(* CODESYS project CtaAppEinsatzDiagramm_2.0.0.0.library
   Description: Einsatzdiagramm Library der CTA
   Version: 2.0.0.0
   Title: CtaAppEinsatzDiagramm
   Author: SIS
   DocFormat: reStructuredText
   LanguageModelAttribute: qualified-access-only
   Placeholder: CtaAppEinsatzDiagramm
   CompiledLibraryCompatibilityVersion: CODESYS V3.5 SP16 Patch 3
   Company: CTA
   DefaultNamespace: CtaAppEinsatzDiagramm

Project tree, tasks and I/O mapping:
  libraries: Standard, 3.5.18.0 (System); CtaAppBmk, 2.0.0.0 (CTA); CtaAppReport, 2.0.0.0 (CTA); CtaSysConfig, 2.0.0.0 (CTA); CtaAppHysterese, 1.0.0.0 (CTA); VisuElemBase, 4.7.0.0 (System); VisuDialogs, * (System); CtaVisSymbols, 2.0.0.0 (CTA); CtaVisUser, 1.0.0.0 (CTA); VisuSymbols, 4.5.0.0 (System); CtaVisApps, 1.0.0.0 (CTA); CtaVisHelp, 1.0.0.0 (CTA)
  40 Visualizations/
    EINSATZGRENZE/
      visualisation VIS_EINSATZGRENZE
      visualisation VIS_EINSATZGRENZE_ITF
      visualisation VIS_EINSATZGRENZE_QUERRY
      DIALOG/
        visualisation DIA_EINSATZGRENZE
        visualisation VIS_DIA_EINSATZGRENZE
        visualisation VIS_DIA_EINSATZGRENZE_ITF
  30 Program Organization Units/
    Einsatzgrenzen/
      function block fbEinsatzgrenze [ST]: actDiagrammPaint, actAktualPoint, actBerrechnung, actÜberwachung, actReport, actConfigFile, proTHIS_REF
  00000000-0000-0000-0000-000000000000|D:\CoDeSys\LibrariesV3\trunk\Intern\CAA\CAA Template\3.4.0.0 draft\Placeholder.xml
  00000000-0000-0000-0000-000000000000|D:\CoDeSys\LibrariesV3\trunk\Intern\CAA\CAA Template\3.2.0.3 draft\Prefix.pdf
  00000000-0000-0000-0000-000000000000|D:\CoDeSys\LibrariesV3\trunk\Intern\CAA\CAA Template\3.5.2.0 draft\Placeholder.xml
  20 Structs/
    Einsatzgrenze/
      data type scParameterEinsatzgrenze
      Paint/
        data type scLinePoint
        data type scDiagrammSizePaint
      Parameter/
        data type scSlopValue1
        data type scSlopValue2
        data type scSlopValue3
        data type scSlopValue4
        data type scSlopValue5
        data type scSlopValue6
        data type scDiagrammSize
        data type scErrorWarning
  50 Images/
  10 Documenation/
    global variables VersionHistory
    global variables readMe
  21 Interface/
    interface ITF_EINSATZGRENZE: proTHIS_REF
  11 Library Parameter/
    global variables Parameter
  12 Konstanten/
    global variables GlobalKonstant
  60 Textlisten/
    text list Error
    text list Info
    text list Warnung
  13 Globale Variablen/
  text list GlobalTextList
  5ce3da45-db07-42e7-a21c-a00fff4ed8f6|C:\Users\sis\Downloads\dip-switch.svg
  5ce3da45-db07-42e7-a21c-a00fff4ed8f6|C:\Users\sis\Downloads\lightning-bolt-circle.svg
  5ce3da45-db07-42e7-a21c-a00fff4ed8f6|C:\Users\sis\Downloads\sine-wave.svg
  5ce3da45-db07-42e7-a21c-a00fff4ed8f6|C:\Users\sis\Downloads\eye.svg
  5ce3da45-db07-42e7-a21c-a00fff4ed8f6|C:\Users\sis\Downloads\lan.svg
*)

// 20 Structs/Einsatzgrenze/scParameterEinsatzgrenze
TYPE scParameterEinsatzgrenze :
    STRUCT
        scDiagrammSize              :   scDiagrammSize;
        fbrMinTc					:	CtaSysConfig.fbREAL;							        // Minimale Kondensationstemperatur [°C] 
        fbrMaxTc					:	CtaSysConfig.fbREAL;							        // Maximale Kondensationstemperatur [°C] 
        fbrMinTo					:	CtaSysConfig.fbREAL;							        // Minimale Verdampfungstemperatur  [°C]
        fbrMaxTo					:	CtaSysConfig.fbREAL; 							        // Maximale Verdampfungstemperatur  [°C]             
        scSlopValue1                :   scSlopValue1;         
        scSlopValue2                :   scSlopValue2;
        scSlopValue3                :   scSlopValue3;
        scSlopValue4                :   scSlopValue4;
        scSlopValue5                :   scSlopValue5;
        scSlopValue6                :   scSlopValue6;        
        scErrorWarning              :   scErrorWarning; 
    END_STRUCT
END_TYPE

// 20 Structs/Einsatzgrenze/Paint/scLinePoint
TYPE scLinePoint :
    STRUCT
        rP1X        :   REAL;
        rP1Y        :   REAL;      
    END_STRUCT
END_TYPE

// 20 Structs/Einsatzgrenze/Paint/scDiagrammSizePaint
TYPE scDiagrammSizePaint :
    STRUCT
        rYMax   :   REAL;
        rYMin   :   REAL;
        rXMax   :   REAL;
        rXMin   :   REAL;    
    END_STRUCT
END_TYPE

// 20 Structs/Einsatzgrenze/Parameter/scSlopValue1
TYPE scSlopValue1 :
    STRUCT
        fbrTcL			    :	CtaSysConfig.fbREAL;							        // Punkt  1 Kompressor-Auslegungsdiagramm [°C] 
        fbrT0L              :   CtaSysConfig.fbREAL;	                                // Punkt  2 Kompressor-Auslegungsdiagramm [°C]
        fbrT0R  		    :	CtaSysConfig.fbREAL;							        // Punkt  3 Kompressor-Auslegungsdiagramm [°C]        
    END_STRUCT
END_TYPE

// 20 Structs/Einsatzgrenze/Parameter/scSlopValue2
TYPE scSlopValue2 :
    STRUCT
        fbrTcR			    :	CtaSysConfig.fbREAL;							        // Punkt  4 Kompressor-Auslegungsdiagramm [°C] 
        fbrT0R  		    :	CtaSysConfig.fbREAL;							        // Punkt  5 Kompressor-Auslegungsdiagramm [°C]        
    END_STRUCT
END_TYPE

// 20 Structs/Einsatzgrenze/Parameter/scSlopValue3
TYPE scSlopValue3 :
    STRUCT
        fbrTcU			    :	CtaSysConfig.fbREAL;							        // Punkt  6 Kompressor-Auslegungsdiagramm [°C] 
    END_STRUCT
END_TYPE

// 20 Structs/Einsatzgrenze/Parameter/scSlopValue4
TYPE scSlopValue4 :
    STRUCT
        fbrTcL			    :	CtaSysConfig.fbREAL;							        // Punkt  7 Kompressor-Auslegungsdiagramm [°C]         
    END_STRUCT
END_TYPE

// 20 Structs/Einsatzgrenze/Parameter/scSlopValue5
TYPE scSlopValue5 :
    STRUCT
        fbrT0L			    :	CtaSysConfig.fbREAL;							        // Punkt  8 Kompressor-Auslegungsdiagramm [°C] 
        fbrT0R  			:	CtaSysConfig.fbREAL;							        // Punkt  9 Kompressor-Auslegungsdiagramm [°C]                
    END_STRUCT
END_TYPE

// 20 Structs/Einsatzgrenze/Parameter/scSlopValue6
TYPE scSlopValue6 :
    STRUCT
        fbrTcO			    :	CtaSysConfig.fbREAL;							        // Punkt 10 Kompressor-Auslegungsdiagramm [°C]                 
    END_STRUCT
END_TYPE

// 20 Structs/Einsatzgrenze/Parameter/scDiagrammSize
TYPE scDiagrammSize :
    STRUCT
        fbrYMax   :   CtaSysConfig.fbREAL;
        fbrYMin   :   CtaSysConfig.fbREAL;
        fbrXMax   :   CtaSysConfig.fbREAL;
        fbrXMin   :   CtaSysConfig.fbREAL;    
    END_STRUCT
END_TYPE

// 20 Structs/Einsatzgrenze/Parameter/scErrorWarning
TYPE scErrorWarning :
    STRUCT
        fbxEnEW1          :   CtaSysConfig.fbBOOL;
        fbxEnEW2          :   CtaSysConfig.fbBOOL;
        fbxEnEW3          :   CtaSysConfig.fbBOOL;
        fbxEnEW4          :   CtaSysConfig.fbBOOL;
        fbxEnEW5          :   CtaSysConfig.fbBOOL;
        fbxEnEW6          :   CtaSysConfig.fbBOOL;
        fbxEnEW7          :   CtaSysConfig.fbBOOL;
        fbtDelayWarning   :   CtaSysConfig.fbTIME;
        fbiAnzError       :   CtaSysConfig.fbINT;
        fbtDelayError     :   CtaSysConfig.fbTIME;
        fbtCountReset     :   CtaSysConfig.fbTIME;
    END_STRUCT
END_TYPE

// 10 Documenation/VersionHistory
(* 

.. image:: ../../Images/CTA_Logo.jpg
   :align: right
   :width: 15% 

**Vorlage**   


============ =========== =========== ============================================
**Date**     **Version** **Author**  **Change**
------------ ----------- ----------- --------------------------------------------
04.03.2021   0.0.0.0     SIS         Vorlage erstellt

============ =========== =========== ============================================


*)
VAR_GLOBAL
    stInfo : STRING:= '0.0.0.0, Vorlage, CTA';
END_VAR

// 10 Documenation/readMe
(*

**ReadMe**
 
|	**Empfehlung**
|
|	Bibliothek CtaAppVerdichter zur Ansteuerung von Verdichtern
|	Instanzieren Sie den CtaAppVerdichter.fbVerdichter in ihrem Funktionsbaustein oder POU beispielsweise als fbVerdiX. (X = Nr.)
|	Instanzieren Sie den CtaAppVerdichter.fbEinsatzgrenze in ihrem Funktionsbaustein oder POU beispielsweise als fbVerdiXEinsatzGr. (X = Nr des Verdicheters)
|	Deklarieren Sie die Struktur Variable welche als Parameter und zur ansteuerung dienen wie im Code beispiel.
|  
| *Beispiel* 

+-----------------------+---------------------------------------------------------------------------------------------------------------------------------------------------------------------------------------------------------------------------------------------------------------------------------------------------------------------------------------------------------------------------------------------------------------------------------------+
| Beschreibung          |  Code                                                                                                                                                                                                                                                                                                                                                                                                                                 |
+=======================+=======================================================================================================================================================================================================================================================================================================================================================================================================================================+
| Pou oder SmFb         | .. code-block:: codesys                                                                                                                                                                                                                                                                                                                                                                                                               |
|                       |                                                                                                                                                                                                                                                                                                                                                                                                                                       |
|                       |	// Deklaration als VAR im POU oder dem selbsterstellten Funktionsbaustein                                                                                                                                                                                                                                                                                                                                                       	|
|                       |   VAR   																																																																																																								|
|						|	    (*Einsatzgrenze Verdichter1*)																																																		 																																															|
|						|		fbVerdi1EinsatzGr	: CtaAppVerdichter.fbEinsatzgrenze;                                                                                                                                                                                                                                                                                                                                                              			|
| 						|	END_VAR                                                                                                                                                                                                                                                                                                                                                                                                                         	|
+-----------------------+---------------------------------------------------------------------------------------------------------------------------------------------------------------------------------------------------------------------------------------------------------------------------------------------------------------------------------------------------------------------------------------------------------------------------------------+
| Code für Init         | .. code-block:: codesys                                                                                                                                                                                                                                                                                                                                                                                                               |
|                       |   																																																																																																									|
| 						|	// Kopieren des nachfolgenden Codes in eine Action zur Initialisierung der Parameter. Zum Beispiel actConfig.																																																																														|
|                       |	{region "Parameter Einsatzgrenzen Verdichter1"}                                                                                                                                                                                                                                                                                                                                                                                     |
| 						|		(*Diagrammgrösse*)																																																																																																				|
|						|		fbVerdi1EinsatzGr.scParaData.scDiagrammSize.fbrYMax               		(_wertInit :=   0.0									, _minInit :=		, _maxInit :=		);		//P1 Diagrammgrösse Y Achse Max																																																						|
|						|		fbVerdi1EinsatzGr.scParaData.scDiagrammSize.fbrYMin						(_wertInit :=   0.0									, _minInit :=		, _maxInit :=		);		//P2 Diagrammgrösse Y Achse Min																																																						|
|						|		fbVerdi1EinsatzGr.scParaData.scDiagrammSize.fbrXMax						(_wertInit :=   0.0									, _minInit :=		, _maxInit :=		);		//P3 Diagrammgrösse X Achse Max																																																						|
|						|		fbVerdi1EinsatzGr.scParaData.scDiagrammSize.fbrXMin						(_wertInit :=   0.0									, _minInit :=		, _maxInit :=		);		//P4 Diagrammgrösse X Achse Min																																																						|
|						|		(*Min Max Tc & To*)																																																		 																																																		|
|						|		fbVerdi1EinsatzGr.scParaData.fbrMinTc									(_wertInit :=   0.0									, _minInit :=		, _maxInit :=		);		//P5 Max Tc																																																											|
|						|		fbVerdi1EinsatzGr.scParaData.fbrMaxTc									(_wertInit :=   0.0									, _minInit :=		, _maxInit :=		);		//P6 Min Tc																																																											|
|						|		fbVerdi1EinsatzGr.scParaData.fbrMinTo									(_wertInit :=   0.0									, _minInit :=		, _maxInit :=		);		//P7 Max To																																																											|
|						|		fbVerdi1EinsatzGr.scParaData.fbrMaxTo									(_wertInit :=   0.0									, _minInit :=		, _maxInit :=		);		//P8 Min To																																																											|
|						|		(*Slop Value 1*)																																																		 																																																		|
|						|		fbVerdi1EinsatzGr.scParaData.scSlopValue1.fbrTcL						(_wertInit :=   0.0									, _minInit :=		, _maxInit :=		);		//P9 Slop Value 1 Tc Links																	    																																					|
|						|		fbVerdi1EinsatzGr.scParaData.scSlopValue1.fbrT0L						(_wertInit :=   0.0									, _minInit :=		, _maxInit :=		);		//P10 Slop Value 1 To Links																												    																										|
|						|		fbVerdi1EinsatzGr.scParaData.scSlopValue1.fbrT0R						(_wertInit :=   0.0									, _minInit :=		, _maxInit :=		);		//P11 Slop Value 1 To Rechts																											    																										|
|						|		(*Slop Value 2*)																																																										 																																	  									|
|						|		fbVerdi1EinsatzGr.scParaData.scSlopValue2.fbrTcR						(_wertInit :=   0.0									, _minInit :=		, _maxInit :=		);		//P12 Slop Value 2 Tc Rechts																    																																					|
|						|		fbVerdi1EinsatzGr.scParaData.scSlopValue2.fbrT0R						(_wertInit :=   0.0									, _minInit :=		, _maxInit :=		);		//P13 Slop Value 2 To Rechts																																								   	 													|
|						|		(*Slop Value 3*)																																																											 																																							    	|
|						|		fbVerdi1EinsatzGr.scParaData.scSlopValue3.fbrTcU						(_wertInit :=   0.0									, _minInit :=		, _maxInit :=		);		//P14 Slop Value 3 Tc Unten																														    																								|
|						|		(*Slop Value 4*)																																																											 																																							    	|
|						|		fbVerdi1EinsatzGr.scParaData.scSlopValue4.fbrTcL						(_wertInit :=   0.0									, _minInit :=		, _maxInit :=		);		//P15 Slop Value 4 Tc Links																																				    																		|
|						|		(*Slop Value 5*)																																																		 																																																		|
|						|		fbVerdi1EinsatzGr.scParaData.scSlopValue5.fbrT0L						(_wertInit :=   0.0									, _minInit :=		, _maxInit :=		);		//P16 Slop Value 5 To Links																																		    																				|
|						|		fbVerdi1EinsatzGr.scParaData.scSlopValue5.fbrT0R						(_wertInit :=   0.0									, _minInit :=		, _maxInit :=		);		//P17 Slop Value 5 To Rechts																																		    																			|
|						|		(*Slop Value 6*)																																																		 																																																		|
|						|		fbVerdi1EinsatzGr.scParaData.scSlopValue6.fbrTcO						(_wertInit :=   0.0									, _minInit :=		, _maxInit :=		);		//P18 Slop Value 6 Tc Oben																																																							|
|						|		(*Error & Warnungen*)																																																																																																		    |
|						|		fbVerdi1EinsatzGr.scParaData.scErrorWarning.fbxEnEW1					(_wertInit := FALSE																			);		//P19 Überwachung Slop Value 1																																	    																				|
|						|		fbVerdi1EinsatzGr.scParaData.scErrorWarning.fbxEnEW2					(_wertInit := FALSE																			);		//P20 Überwachung Slop Value 2																																										    											|
|						|		fbVerdi1EinsatzGr.scParaData.scErrorWarning.fbxEnEW3					(_wertInit := FALSE																			);		//P21 Überwachung Slop Value 3																														   																								|
|						|		fbVerdi1EinsatzGr.scParaData.scErrorWarning.fbxEnEW4					(_wertInit := FALSE																			);		//P22 Überwachung Slop Value 4																																								    													|
|						|		fbVerdi1EinsatzGr.scParaData.scErrorWarning.fbxEnEW5					(_wertInit := FALSE																			);		//P23 Überwachung Slop Value 5				   																																																		|
|						|		fbVerdi1EinsatzGr.scParaData.scErrorWarning.fbxEnEW6					(_wertInit := FALSE																			);		//P24 Überwachung Slop Value 6																						   																																|
|						|		fbVerdi1EinsatzGr.scParaData.scErrorWarning.fbxEnEW7					(_wertInit := FALSE																			);		//P25 Überwachung Slop Value 7														    																																							|
|						|		fbVerdi1EinsatzGr.scParaData.scErrorWarning.fbtDelayWarning				(_wertInit := T#00S									, _minInit :=		, _maxInit :=		);		//P26 Warnungsverzögerung																																																							|
|						|		fbVerdi1EinsatzGr.scParaData.scErrorWarning.fbiAnzError					(_wertInit :=     0									, _minInit :=		, _maxInit :=		);		//P27 Anzahl Error Autoquittierungen																																																				|
|						|		fbVerdi1EinsatzGr.scParaData.scErrorWarning.fbtDelayError				(_wertInit := T#00S									, _minInit :=	    , _maxInit :=		);		//P28 Errorverzögerung																																																								|
|						|		fbVerdi1EinsatzGr.scParaData.scErrorWarning.fbtCountReset				(_wertInit := T#00S									, _minInit :=		, _maxInit :=		);		//P29 Reset des Zähler nach t																																																						|
|						|	{endregion}                                             	                                                                                                         																																																																|
+-----------------------+---------------------------------------------------------------------------------------------------------------------------------------------------------------------------------------------------------------------------------------------------------------------------------------------------------------------------------------------------------------------------------------------------------------------------------------+
*)                                                                                                                                                                                                                                                                                                                                                                                                                                                               
 VAR_GLOBAL                                                                                                                                                                                                                                                                                                                                                                                                                                                      
    xReadMeDone              :   BOOL;                                                                                                                                                                                                                                                                                                                                                                                                                           
END_VAR

// 11 Library Parameter/Parameter
{attribute 'qualified_only'}
VAR_GLOBAL CONSTANT
    iMaxVerdichter :   INT   := 60;         // Maximale Anzahl verwendeter AT-Bausteine    
END_VAR

// 12 Konstanten/GlobalKonstant
{attribute 'qualified_only'}
VAR_GLOBAL CONSTANT 	
	stReportTextListError   : CtaAppReport.stReportTextList := 'CtaAppEinsatzDiagramm.Error';
	stReportTextListWarning : CtaAppReport.stReportTextList := 'CtaAppEinsatzDiagramm.Warnung';
	stReportTextListInfo    : CtaAppReport.stReportTextList := 'CtaAppEinsatzDiagramm.Info';	
END_VAR

// 30 Program Organization Units/Einsatzgrenzen/fbEinsatzgrenze
FUNCTION_BLOCK fbEinsatzgrenze IMPLEMENTS ITF_EINSATZGRENZE
VAR_INPUT
	xEnable							:	BOOL;
	rtcAct						    :	REAL;							        // Aktuelle Kondensationstemperatur [°C] 
	rt0Act						    :	REAL;							        // Aktuelle Verdampfungstemperatur [°C]  
	ITF_BMK							:	CtaAppBmk.ITF_BMK;
    ITF_REPORTMANAGER     			:   CtaAppReport.ITF_REPORTMANAGER;
END_VAR                           
VAR
    scParaData                      :   scParameterEinsatzgrenze;
    scDiagrammSizePaint             :   scDiagrammSizePaint;
    xInitDone                       :   BOOL;
    ayDiagramm                      :   ARRAY[1..14] OF scLinePoint;
    ayAktualPoint                   :   ARRAY[1..60] OF scLinePoint;
    TON_TRIG_SAVE_FAST              :   TON;
    TON_TRIG_SAVE                   :   TON;    
    iFor                            :   INT;
	diFor                           :   DINT;
    iSel                            :   INT;
    rTempCalc1                      :   REAL;
    rTempCalc2                      :   REAL;    
    rMaxTcL                         :   REAL;
    rMaxTcR                         :   REAL;
    rMinTcR                         :   REAL;
    ayTcMax                         :   ARRAY[1..2] OF scLinePoint;
    ayTcMin                         :   ARRAY[1..2] OF scLinePoint;
    fbHystereseDMO1                 :   CtaAppHysterese.fbHyst_Dir;    
    fbHystereseDRO2                 :   CtaAppHysterese.fbHyst_Dir;  
    fbHystereseDMR3                 :   CtaAppHysterese.fbHyst_Dir;      
    fbHystereseRRU4                 :   CtaAppHysterese.fbHyst_Rev;  
    fbHystereseRMU5                 :   CtaAppHysterese.fbHyst_Rev; 
    fbHystereseRLM6                 :   CtaAppHysterese.fbHyst_Rev; 
    fbHystereseDLO7                 :   CtaAppHysterese.fbHyst_Dir;     
    // Configfile Manager
    fbConfigFile                    :   CtaSysConfig.fbConfigFile;  
    // Error Code Baustein	
	ayErrorReporter					:	ARRAY[11..17] OF CtaAppReport.fbReporter;
	ayWarningReporter				:	ARRAY[11..17] OF CtaAppReport.fbReporter; 
END_VAR

(* Parameter *)
actConfigFile();
(* Diagramm paint *)
actDiagrammPaint();
(* Point Actualisation *)
actAktualPoint();
(* Berrechnung Einstzgrenzen *)
actBerrechnung();
(* Überachung einsatzgrenzen *)
actÜberwachung();
(* Reports *)
IF __QUERYINTERFACE(ITF_REPORTMANAGER,ITF_REPORTMANAGER) AND __QUERYINTERFACE(ITF_BMK,ITF_BMK) THEN
	actReport();
END_IF;

ACTION actDiagrammPaint:
IF fbConfigFile.proEventDetekted THEN
    // Diagramm grösse
    scDiagrammSizePaint.rXMin   := scParaData.scdiagrammSize.fbrXMin.provalue;
    scDiagrammSizePaint.rXMax   := scParaData.scdiagrammSize.fbrXMax.provalue;
    scDiagrammSizePaint.rYMin   := scParaData.scdiagrammSize.fbrYMin.provalue;
    scDiagrammSizePaint.rYMax   := scParaData.scdiagrammSize.fbrYMax.provalue;
    
    // Punkt 1 Links Horizontal Oben
    ayDiagramm[1].rP1X  := scParaData.scSlopValue1.fbrT0L.provalue;
    ayDiagramm[1].rP1Y  := scParaData.scSlopValue1.fbrTcL.provalue;
    ayDiagramm[2].rP1X  := scParaData.scSlopValue1.fbrT0R.provalue;
    ayDiagramm[2].rP1Y  := scParaData.scSlopValue1.fbrTcL.provalue;
    // Punkt 2 Schräg rechts Oben
    ayDiagramm[3].rP1X  := ayDiagramm[2].rP1X;
    ayDiagramm[3].rP1Y  := ayDiagramm[2].rP1Y;
    ayDiagramm[4].rP1X  := scParaData.scSlopValue2.fbrT0R.provalue;
    ayDiagramm[4].rP1Y  := scParaData.scSlopValue2.fbrTcR.provalue;
    // Punkt 3 Vertikal rechts
    ayDiagramm[5].rP1X  := ayDiagramm[4].rP1X;
    ayDiagramm[5].rP1Y  := ayDiagramm[4].rP1Y;
    ayDiagramm[6].rP1X  := ayDiagramm[4].rP1X;
    ayDiagramm[6].rP1Y  := scParaData.scSlopValue3.fbrTcU.proValue;
    // Punkt 4 Schräg rechts Unten
    ayDiagramm[7].rP1X  := ayDiagramm[6].rP1X;
    ayDiagramm[7].rP1Y  := ayDiagramm[6].rP1Y;
    ayDiagramm[8].rP1X  := scParaData.scSlopValue5.fbrT0R.proValue;
    ayDiagramm[8].rP1Y  := scParaData.scSlopValue4.fbrTcL.proValue;
    // Punkt 5 Horizontal Unten
    ayDiagramm[9].rP1X  := ayDiagramm[8].rP1X;
    ayDiagramm[9].rP1Y  := ayDiagramm[8].rP1Y;
    ayDiagramm[10].rP1X  := scParaData.scSlopValue5.fbrT0L.proValue;
    ayDiagramm[10].rP1Y  := scParaData.scSlopValue4.fbrTcL.proValue;
    // Punkt 6 Vertikal Links
    ayDiagramm[11].rP1X  := ayDiagramm[10].rP1X;
    ayDiagramm[11].rP1Y  := ayDiagramm[10].rP1Y;
    ayDiagramm[12].rP1X  := ayDiagramm[10].rP1X;
    ayDiagramm[12].rP1Y  := scParaData.scSlopValue6.fbrTcO.proValue;
    // Punkt 7 Schräg Links Oben
    ayDiagramm[13].rP1X  := ayDiagramm[12].rP1X;
    ayDiagramm[13].rP1Y  := ayDiagramm[12].rP1Y;
    ayDiagramm[14].rP1X  := ayDiagramm[1].rP1X;
    ayDiagramm[14].rP1Y  := ayDiagramm[1].rP1Y;
    // TcMax
    ayTcMax[1].rP1X := scParaData.scDiagrammSize.fbrXMax.proValue;
    ayTcMax[1].rP1Y := scParaData.fbrMaxTc.proValue;
    ayTcMax[2].rP1X := scParaData.scDiagrammSize.fbrXMin.proValue;
    ayTcMax[2].rP1Y := scParaData.fbrMaxTc.proValue;
    // TcMin
    ayTcMin[1].rP1X := scParaData.scDiagrammSize.fbrXMax.proValue;
    ayTcMin[1].rP1Y := scParaData.fbrMinTc.proValue;
    ayTcMin[2].rP1X := scParaData.scDiagrammSize.fbrXMin.proValue;
    ayTcMin[2].rP1Y := scParaData.fbrMinTc.proValue;
END_IF;
END_ACTION

ACTION actAktualPoint:
TON_TRIG_SAVE       (IN := NOT TON_TRIG_SAVE.Q , PT := T#1S100MS);
TON_TRIG_SAVE_FAST  (IN := NOT TON_TRIG_SAVE.Q , PT := T#1S);
IF xEnable THEN
    IF NOT xInitDone THEN
        FOR iFor := 60 TO 1 BY -1 DO
            // Aktuelle Position
            ayAktualPoint[iFor].rP1X := rt0Act;
            ayAktualPoint[iFor].rP1Y := rtcAct;     
        END_FOR;   
        xInitDone   := TRUE;   
    ELSE
        IF ayAktualPoint[1].rP1X <> rt0Act OR ayAktualPoint[1].rP1Y <> rtcAct THEN
                // Aktuelle Position
                ayAktualPoint[1].rP1X := rt0Act;
                ayAktualPoint[1].rP1Y := rtcAct;
        END_IF;
        IF TON_TRIG_SAVE.Q THEN
            FOR iFor := 60 TO 10 BY -1 DO
                ayAktualPoint[iFor].rP1X := ayAktualPoint[iFor-1].rP1X;
                ayAktualPoint[iFor].rP1Y := ayAktualPoint[iFor-1].rP1Y;         
            END_FOR;
        END_IF;  
        IF TON_TRIG_SAVE_FAST.Q THEN
            FOR iFor := 10 TO 2 BY -1 DO
                ayAktualPoint[iFor].rP1X := ayAktualPoint[iFor-1].rP1X;
                ayAktualPoint[iFor].rP1Y := ayAktualPoint[iFor-1].rP1Y;         
            END_FOR;
        END_IF;                   
    END_IF;
ELSE
    FOR iFor := 1 TO 60 DO
        ayAktualPoint[iFor].rP1X   := 0; 
	    ayAktualPoint[iFor].rP1Y   := 0;
    END_FOR;
    xInitDone := FALSE;
END_IF
END_ACTION

ACTION actBerrechnung:
// Tc Max Links
IF (ayDiagramm[13].rP1X-ayDiagramm[14].rP1X) <> 0 THEN
    rTempCalc1  := ((ayDiagramm[13].rP1Y-ayDiagramm[14].rP1Y)/(ayDiagramm[13].rP1X-ayDiagramm[14].rP1X));   
    rTempCalc2  := ayDiagramm[13].rP1Y-rTempCalc1*ayDiagramm[13].rP1X; 
    rMaxTcL     := LIMIT(scParaData.fbrMinTc.proValue,(rt0Act * rTempCalc1 +rTempCalc2),scParaData.fbrMaxTc.proValue);
ELSE
	rMaxTcL		:= LIMIT(scParaData.fbrMinTc.proValue,ayDiagramm[13].rP1Y,scParaData.fbrMaxTc.proValue);
END_IF;
// Tc Max Rechts
IF (ayDiagramm[3].rP1X-ayDiagramm[4].rP1X) <> 0 THEN
    rTempCalc1  := ((ayDiagramm[3].rP1Y-ayDiagramm[4].rP1Y)/(ayDiagramm[3].rP1X-ayDiagramm[4].rP1X));   
    rTempCalc2  := ayDiagramm[3].rP1Y-rTempCalc1*ayDiagramm[3].rP1X; 
    rMaxTcR     := LIMIT(scParaData.fbrMinTc.proValue,(rt0Act * rTempCalc1 +rTempCalc2),scParaData.fbrMaxTc.proValue);
ELSE
	rMaxTcR     := LIMIT(scParaData.fbrMinTc.proValue,(ayDiagramm[3].rP1Y),scParaData.fbrMaxTc.proValue);
END_IF;
// Tc Min Rechts
IF (ayDiagramm[7].rP1X-ayDiagramm[8].rP1X) <> 0 THEN
    rTempCalc1  := ((ayDiagramm[7].rP1Y-ayDiagramm[8].rP1Y)/(ayDiagramm[7].rP1X-ayDiagramm[8].rP1X));   
    rTempCalc2  := ayDiagramm[7].rP1Y-rTempCalc1*ayDiagramm[7].rP1X; 
    rMinTcR     := LIMIT(scParaData.fbrMinTc.proValue,(rt0Act * rTempCalc1 +rTempCalc2),scParaData.fbrMaxTc.proValue);
ELSE
	rMinTcR		:= LIMIT(scParaData.fbrMinTc.proValue,ayDiagramm[7].rP1Y,scParaData.fbrMaxTc.proValue);
END_IF;
END_ACTION

ACTION actÜberwachung:
// Diagramm mitte oben Nr 1
fbHystereseDMO1(    rIn        :=  rtcAct,
                    rSet       :=  scParaData.fbrMaxTc.proValue,
                    rDiffOn    :=  0,
                    rDIffOff   :=  0.5);

// Diagramm rechts oben Nr 2
fbHystereseDRO2(    rIn        :=  rtcAct,
                    rSet       :=  rMaxTcR,
                    rDiffOn    :=  0,
                    rDIffOff   :=  0.5);
                    
// Diagramm mittte rechts Nr 3
fbHystereseDMR3(    rIn        :=  rt0Act,
                    rSet       :=  scParaData.fbrMaxTo.proValue,
                    rDiffOn    :=  0,
                    rDIffOff   :=  0.5);
                    
// Diagramm rechts unten Nr 4                
fbHystereseRRU4(    rIn        :=  rtcAct,
                    rSet       :=  rMinTcR,
                    rDiffOn    :=  0,
                    rDIffOff   :=  0.5);      

// Diagramm mitte unten Nr 5                
fbHystereseRMU5(    rIn        :=  rtcAct,
                    rSet       :=  scParaData.fbrMinTc.proValue,
                    rDiffOn    :=  0,
                    rDIffOff   :=  0.5);    
                    
// Diagramm links mitte Nr 6                
fbHystereseRLM6(    rIn        :=  rt0Act,
                    rSet       :=  scParaData.fbrMinTo.proValue,
                    rDiffOn    :=  0,
                    rDIffOff   :=  0.5);  
     
// Diagramm links oben Nr 7
fbHystereseDLO7(    rIn        :=  rtcAct,
                    rSet       :=  rMaxTcL,
                    rDiffOn    :=  0,
                    rDIffOff   :=  0.5);
END_ACTION

ACTION actReport:
(* Warnungen *)                       
        (* Meldung Diagramm überschritten 11*)
        ayWarningReporter[11].proPrio := 1;    
		ayWarningReporter[11].metReport(		xSetReportIn					:= scParaData.scErrorWarning.fbxEnEW1.proValue AND fbHystereseDMO1.xOut AND xEnable,
												iReportID						:= 11,
												enReportTypeIn					:= CtaAppReport.enReportType.Warning,  
												enReportAcknowledgeTypeIn   	:= CtaAppReport.enReportAcknowledgeType.Auto,
												tDelay							:= scParaData.scErrorWarning.fbtDelayWarning.proValue, 
												ITF_BMK_IN						:= ITF_BMK,			              
												pstReportTextListIn				:= ADR(GlobalKonstant.stReportTextListWarning),
												stOptionalReportText		    := '',   
												iRetryTilReportLock 		    := 0, 
												xResetCount         		    := FALSE,  
												tReset						    := T#0S);    		
                                        
        (* Meldung Diagramm überschritten 12*)   
        ayWarningReporter[12].proPrio := 1;       
		ayWarningReporter[12].metReport(		xSetReportIn					:= scParaData.scErrorWarning.fbxEnEW2.proValue AND fbHystereseDRO2.xOut AND NOT fbHystereseDMO1.xOut AND xEnable,
												iReportID						:= 12,
												enReportTypeIn					:= CtaAppReport.enReportType.Warning,  
												enReportAcknowledgeTypeIn   	:= CtaAppReport.enReportAcknowledgeType.Auto,
												tDelay							:= scParaData.scErrorWarning.fbtDelayWarning.proValue, 
												ITF_BMK_IN						:= ITF_BMK,			              
												pstReportTextListIn				:= ADR(GlobalKonstant.stReportTextListWarning),
												stOptionalReportText		    := '',   
												iRetryTilReportLock 		    := 0, 
												xResetCount         		    := FALSE,  
												tReset						    := T#0S);                            
                                        
        (* Meldung Diagramm überschritten 13*)  
        ayWarningReporter[13].proPrio := 1;     
		ayWarningReporter[13].metReport(		xSetReportIn					:= scParaData.scErrorWarning.fbxEnEW3.proValue AND fbHystereseDMR3.xOut AND xEnable,
												iReportID						:= 13,
												enReportTypeIn					:= CtaAppReport.enReportType.Warning,  
												enReportAcknowledgeTypeIn   	:= CtaAppReport.enReportAcknowledgeType.Auto,
												tDelay							:= scParaData.scErrorWarning.fbtDelayWarning.proValue, 
												ITF_BMK_IN						:= ITF_BMK,			              
												pstReportTextListIn				:= ADR(GlobalKonstant.stReportTextListWarning),
												stOptionalReportText		    := '',   
												iRetryTilReportLock 		    := 0, 
												xResetCount         		    := FALSE,  
												tReset						    := T#0S);        
                                        
        (* Meldung Diagramm überschritten 14*) 
        ayWarningReporter[14].proPrio := 1;        
		ayWarningReporter[14].metReport(		xSetReportIn					:= scParaData.scErrorWarning.fbxEnEW4.proValue AND fbHystereseRRU4.xOut AND NOT fbHystereseRMU5.xOut AND xEnable,
												iReportID						:= 14,
												enReportTypeIn					:= CtaAppReport.enReportType.Warning,  
												enReportAcknowledgeTypeIn   	:= CtaAppReport.enReportAcknowledgeType.Auto,
												tDelay							:= scParaData.scErrorWarning.fbtDelayWarning.proValue, 
												ITF_BMK_IN						:= ITF_BMK,			              
												pstReportTextListIn				:= ADR(GlobalKonstant.stReportTextListWarning),
												stOptionalReportText		    := '',   
												iRetryTilReportLock 		    := 0, 
												xResetCount         		    := FALSE,  
												tReset						    := T#0S);                                    
                                
        (* Meldung Diagramm überschritten 15*)  
        ayWarningReporter[15].proPrio := 1;           
		ayWarningReporter[15].metReport(		xSetReportIn					:= scParaData.scErrorWarning.fbxEnEW5.proValue AND fbHystereseRMU5.xOut AND xEnable,
												iReportID						:= 15,
												enReportTypeIn					:= CtaAppReport.enReportType.Warning,  
												enReportAcknowledgeTypeIn   	:= CtaAppReport.enReportAcknowledgeType.Auto,
												tDelay							:= scParaData.scErrorWarning.fbtDelayWarning.proValue, 
												ITF_BMK_IN						:= ITF_BMK,			              
												pstReportTextListIn				:= ADR(GlobalKonstant.stReportTextListWarning),
												stOptionalReportText		    := '',   
												iRetryTilReportLock 		    := 0, 
												xResetCount         		    := FALSE,  
												tReset						    := T#0S);                        
      
        (* Meldung Diagramm überschritten 16*)  
        ayWarningReporter[16].proPrio := 1;                        
		ayWarningReporter[16].metReport(		xSetReportIn					:= scParaData.scErrorWarning.fbxEnEW6.proValue AND fbHystereseRLM6.xOut AND xEnable,
												iReportID						:= 16,
												enReportTypeIn					:= CtaAppReport.enReportType.Warning,  
												enReportAcknowledgeTypeIn   	:= CtaAppReport.enReportAcknowledgeType.Auto,
												tDelay							:= scParaData.scErrorWarning.fbtDelayWarning.proValue, 
												ITF_BMK_IN						:= ITF_BMK,			              
												pstReportTextListIn				:= ADR(GlobalKonstant.stReportTextListWarning),
												stOptionalReportText		    := '',   
												iRetryTilReportLock 		    := 0, 
												xResetCount         		    := FALSE,  
												tReset						    := T#0S);            
                                        
        (* Meldung Diagramm überschritten 17*)  
        ayWarningReporter[17].proPrio := 1;     
		ayWarningReporter[17].metReport(		xSetReportIn					:= scParaData.scErrorWarning.fbxEnEW7.proValue AND fbHystereseDLO7.xOut AND NOT fbHystereseDMO1.xOut AND xEnable,
												iReportID						:= 17,
												enReportTypeIn					:= CtaAppReport.enReportType.Warning,  
												enReportAcknowledgeTypeIn   	:= CtaAppReport.enReportAcknowledgeType.Auto,
												tDelay							:= scParaData.scErrorWarning.fbtDelayWarning.proValue, 
												ITF_BMK_IN						:= ITF_BMK,			              
												pstReportTextListIn				:= ADR(GlobalKonstant.stReportTextListWarning),
												stOptionalReportText		    := '',   
												iRetryTilReportLock 		    := 0, 
												xResetCount         		    := FALSE,  
												tReset						    := T#0S);                          
        
(* Störungen *)
        (* Meldung Diagramm überschritten 11*)
        ayErrorReporter[11].proPrio := 1;   
		ayErrorReporter[11].metReport(			xSetReportIn					:= scParaData.scErrorWarning.fbxEnEW1.proValue AND fbHystereseDMO1.xOut AND xEnable,
												iReportID						:= 11,
												enReportTypeIn					:= CtaAppReport.enReportType.Error,  
												enReportAcknowledgeTypeIn   	:= CtaAppReport.enReportAcknowledgeType.RetryN,
												tDelay							:= scParaData.scErrorWarning.fbtDelayError.proValue, 
												ITF_BMK_IN						:= ITF_BMK,			              
												pstReportTextListIn				:= ADR(GlobalKonstant.stReportTextListError),
												stOptionalReportText		    := '',   
												iRetryTilReportLock 		    := scParaData.scErrorWarning.fbiAnzError.proValue, 
												xResetCount         		    := FALSE,  
												tReset						    := scParaData.scErrorWarning.fbtCountReset.proValue); 	
	                                       
        (* Meldung Diagramm überschritten 12*) 
        ayErrorReporter[12].proPrio := 1;   
		ayErrorReporter[12].metReport(			xSetReportIn					:= scParaData.scErrorWarning.fbxEnEW2.proValue AND fbHystereseDRO2.xOut AND NOT fbHystereseDMO1.xOut AND xEnable,
												iReportID						:= 12,
												enReportTypeIn					:= CtaAppReport.enReportType.Error,  
												enReportAcknowledgeTypeIn   	:= CtaAppReport.enReportAcknowledgeType.RetryN,
												tDelay							:= scParaData.scErrorWarning.fbtDelayError.proValue, 
												ITF_BMK_IN						:= ITF_BMK,			              
												pstReportTextListIn				:= ADR(GlobalKonstant.stReportTextListError),
												stOptionalReportText		    := '',   
												iRetryTilReportLock 		    := scParaData.scErrorWarning.fbiAnzError.proValue, 
												xResetCount         		    := FALSE,  
												tReset						    := scParaData.scErrorWarning.fbtCountReset.proValue);                              

                                        
        (* Meldung Diagramm überschritten 13*) 
        ayErrorReporter[13].proPrio := 1;       
		ayErrorReporter[13].metReport(			xSetReportIn					:= scParaData.scErrorWarning.fbxEnEW3.proValue AND fbHystereseDMR3.xOut AND xEnable,
												iReportID						:= 13,
												enReportTypeIn					:= CtaAppReport.enReportType.Error,  
												enReportAcknowledgeTypeIn   	:= CtaAppReport.enReportAcknowledgeType.RetryN,
												tDelay							:= scParaData.scErrorWarning.fbtDelayError.proValue, 
												ITF_BMK_IN						:= ITF_BMK,			              
												pstReportTextListIn				:= ADR(GlobalKonstant.stReportTextListError),
												stOptionalReportText		    := '',   
												iRetryTilReportLock 		    := scParaData.scErrorWarning.fbiAnzError.proValue, 
												xResetCount         		    := FALSE,  
												tReset						    := scParaData.scErrorWarning.fbtCountReset.proValue);    
                                        
        (* Meldung Diagramm überschritten 14*)     
        ayErrorReporter[14].proPrio := 1;      
		ayErrorReporter[14].metReport(			xSetReportIn					:= scParaData.scErrorWarning.fbxEnEW4.proValue AND fbHystereseRRU4.xOut AND NOT fbHystereseRMU5.xOut AND xEnable,
												iReportID						:= 14,
												enReportTypeIn					:= CtaAppReport.enReportType.Error,  
												enReportAcknowledgeTypeIn   	:= CtaAppReport.enReportAcknowledgeType.RetryN,
												tDelay							:= scParaData.scErrorWarning.fbtDelayError.proValue, 
												ITF_BMK_IN						:= ITF_BMK,			              
												pstReportTextListIn				:= ADR(GlobalKonstant.stReportTextListError),
												stOptionalReportText		    := '',   
												iRetryTilReportLock 		    := scParaData.scErrorWarning.fbiAnzError.proValue, 
												xResetCount         		    := FALSE,  
												tReset						    := scParaData.scErrorWarning.fbtCountReset.proValue);                              
                                
        (* Meldung Diagramm überschritten 5*)  
        ayErrorReporter[15].proPrio := 1;   
		ayErrorReporter[15].metReport(			xSetReportIn					:= scParaData.scErrorWarning.fbxEnEW5.proValue AND fbHystereseRMU5.xOut AND xEnable,
												iReportID						:= 15,
												enReportTypeIn					:= CtaAppReport.enReportType.Error,  
												enReportAcknowledgeTypeIn   	:= CtaAppReport.enReportAcknowledgeType.RetryN,
												tDelay							:= scParaData.scErrorWarning.fbtDelayError.proValue, 
												ITF_BMK_IN						:= ITF_BMK,			              
												pstReportTextListIn				:= ADR(GlobalKonstant.stReportTextListError),
												stOptionalReportText		    := '',   
												iRetryTilReportLock 		    := scParaData.scErrorWarning.fbiAnzError.proValue, 
												xResetCount         		    := FALSE,  
												tReset						    := scParaData.scErrorWarning.fbtCountReset.proValue);                             
      
        (* Meldung Diagramm überschritten 16*) 
        ayErrorReporter[16].proPrio := 1;   
		ayErrorReporter[16].metReport(			xSetReportIn					:= scParaData.scErrorWarning.fbxEnEW6.proValue AND fbHystereseRLM6.xOut AND xEnable,
												iReportID						:= 16,
												enReportTypeIn					:= CtaAppReport.enReportType.Error,  
												enReportAcknowledgeTypeIn   	:= CtaAppReport.enReportAcknowledgeType.RetryN,
												tDelay							:= scParaData.scErrorWarning.fbtDelayError.proValue, 
												ITF_BMK_IN						:= ITF_BMK,			              
												pstReportTextListIn				:= ADR(GlobalKonstant.stReportTextListError),
												stOptionalReportText		    := '',   
												iRetryTilReportLock 		    := scParaData.scErrorWarning.fbiAnzError.proValue, 
												xResetCount         		    := FALSE,  
												tReset						    := scParaData.scErrorWarning.fbtCountReset.proValue);                                
                                        
        (* Meldung Diagramm überschritten 17*) 
        ayErrorReporter[17].proPrio := 1;     
		ayErrorReporter[17].metReport(			xSetReportIn					:= scParaData.scErrorWarning.fbxEnEW7.proValue AND fbHystereseDLO7.xOut AND NOT fbHystereseDMO1.xOut AND xEnable,
												iReportID						:= 17,
												enReportTypeIn					:= CtaAppReport.enReportType.Error,  
												enReportAcknowledgeTypeIn   	:= CtaAppReport.enReportAcknowledgeType.RetryN,
												tDelay							:= scParaData.scErrorWarning.fbtDelayError.proValue, 
												ITF_BMK_IN						:= ITF_BMK,			              
												pstReportTextListIn				:= ADR(GlobalKonstant.stReportTextListError),
												stOptionalReportText		    := '',   
												iRetryTilReportLock 		    := scParaData.scErrorWarning.fbiAnzError.proValue, 
												xResetCount         		    := FALSE,  
												tReset						    := scParaData.scErrorWarning.fbtCountReset.proValue);                           
                                  
(* Sync Reports *)                                         
FOR difor := LOWER_BOUND(ayErrorReporter,1) TO UPPER_BOUND(ayErrorReporter,1) DO
	ITF_REPORTMANAGER.metSyncReporter(ayErrorReporter[difor]);	
END_FOR;
FOR difor := LOWER_BOUND(ayWarningReporter,1) TO UPPER_BOUND(ayWarningReporter,1) DO
	ITF_REPORTMANAGER.metSyncReporter(ayWarningReporter[difor]);	
END_FOR;
END_ACTION

ACTION actConfigFile:
// Aufruf fbConfigFile
fbConfigFile();
(* Diagramm Grösse *)
scParaData.scDiagrammSize.fbrYMax         ( _usiParaNr :=  1, itfConfigFb := fbconfigFile );    
scParaData.scDiagrammSize.fbrYMin         ( _usiParaNr :=  2, itfConfigFb := fbconfigFile );
scParaData.scDiagrammSize.fbrXMax         ( _usiParaNr :=  3, itfConfigFb := fbconfigFile );
scParaData.scDiagrammSize.fbrXMin         ( _usiParaNr :=  4, itfConfigFb := fbconfigFile );
(* Min Max Tc & To *)                                        
scParaData.fbrMinTc                       ( _usiParaNr :=  5, itfConfigFb := fbconfigFile );
scParaData.fbrMaxTc                       ( _usiParaNr :=  6, itfConfigFb := fbconfigFile );
scParaData.fbrMinTo                       ( _usiParaNr :=  7, itfConfigFb := fbconfigFile );
scParaData.fbrMaxTo                       ( _usiParaNr :=  8, itfConfigFb := fbconfigFile );
(* Slop Value 1 *)                                           
scParaData.scSlopValue1.fbrTcL            ( _usiParaNr :=  9, itfConfigFb := fbconfigFile );
scParaData.scSlopValue1.fbrT0L            ( _usiParaNr := 10, itfConfigFb := fbconfigFile );
scParaData.scSlopValue1.fbrT0R            ( _usiParaNr := 11, itfConfigFb := fbconfigFile );
(* Slop Value 2 *)                                           
ScParaData.scSlopValue2.fbrTcR            ( _usiParaNr := 12, itfConfigFb := fbconfigFile );
ScParaData.scSlopValue2.fbrT0R            ( _usiParaNr := 13, itfConfigFb := fbconfigFile );
(* Slop Value 3 *)                                           
scParaData.scSlopValue3.fbrTcU            ( _usiParaNr := 14, itfConfigFb := fbconfigFile );        
(* Slop Value 4 *)                                           
scParaData.scSlopValue4.fbrTcL            ( _usiParaNr := 15, itfConfigFb := fbconfigFile );   
(* Slop Value 5 *)                                           
scParaData.scSlopValue5.fbrT0L            ( _usiParaNr := 16, itfConfigFb := fbconfigFile );     
scParaData.scSlopValue5.fbrT0R            ( _usiParaNr := 17, itfConfigFb := fbconfigFile );     
(* Slop Value 6 *)                                           
scParaData.scSlopValue6.fbrTcO            ( _usiParaNr := 18, itfConfigFb := fbconfigFile );                      
(* Error & Warnungen *)                                      
scparaData.scErrorWarning.fbxEnEW1        ( _usiParaNr := 19, itfConfigFb := fbconfigFile );            
scparaData.scErrorWarning.fbxEnEW2        ( _usiParaNr := 20, itfConfigFb := fbconfigFile );
scparaData.scErrorWarning.fbxEnEW3        ( _usiParaNr := 21, itfConfigFb := fbconfigFile );
scparaData.scErrorWarning.fbxEnEW4        ( _usiParaNr := 22, itfConfigFb := fbconfigFile );
scparaData.scErrorWarning.fbxEnEW5        ( _usiParaNr := 23, itfConfigFb := fbconfigFile );
scparaData.scErrorWarning.fbxEnEW6        ( _usiParaNr := 24, itfConfigFb := fbconfigFile );
scparaData.scErrorWarning.fbxEnEW7        ( _usiParaNr := 25, itfConfigFb := fbconfigFile );
scparaData.scErrorWarning.fbtDelayWarning ( _usiParaNr := 26, itfConfigFb := fbconfigFile );
scparaData.scErrorWarning.fbiAnzError     ( _usiParaNr := 27, itfConfigFb := fbconfigFile );
scparaData.scErrorWarning.fbtDelayError   ( _usiParaNr := 28, itfConfigFb := fbconfigFile );
scparaData.scErrorWarning.fbtCountReset   ( _usiParaNr := 29, itfConfigFb := fbconfigFile );
END_ACTION

PROPERTY proTHIS_REF : REFERENCE TO fbEinsatzgrenze
GET
proTHIS_REF REF= THIS^;
END_GET
END_PROPERTY

END_FUNCTION_BLOCK

// 21 Interface/ITF_EINSATZGRENZE
INTERFACE ITF_EINSATZGRENZE EXTENDS __SYSTEM.IQueryInterface

PROPERTY proTHIS_REF : REFERENCE TO fbEinsatzgrenze
GET
END_GET
END_PROPERTY

END_INTERFACE

// 40 Visualizations/EINSATZGRENZE/VIS_EINSATZGRENZE
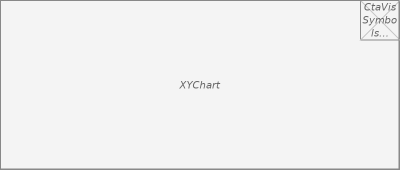
VISUALIZATION VIS_EINSATZGRENZE  // 400x170
VAR_INPUT
    {attribute 'initialize_on_call'}
    ITF_EINSATZGRENZEIn : ITF_EINSATZGRENZE;	
END_VAR
    Frame (0,0 400x170), invisible if: NOT __QUERYINTERFACE(ITF_EINSATZGRENZEIn,ITF_EINSATZGRENZEIn)
        shows VIS_EINSATZGRENZE_QUERRY(ITF_EINSATZGRENZEIn := ITF_EINSATZGRENZEIn)
END_VISUALIZATION

// 40 Visualizations/EINSATZGRENZE/DIALOG/DIA_EINSATZGRENZE
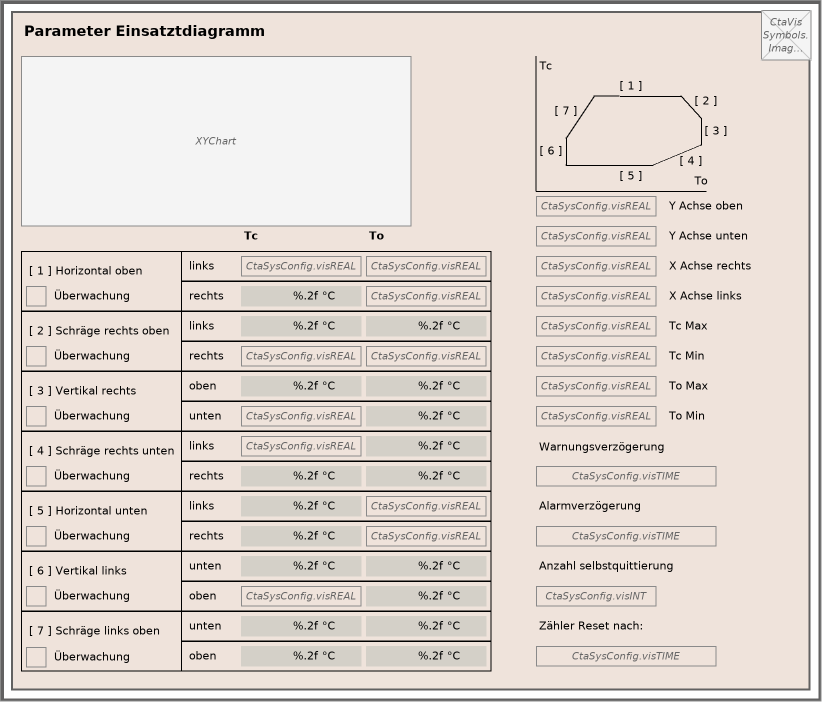
VISUALIZATION DIA_EINSATZGRENZE  // 822x702
VAR_INPUT
    ITF_EINSATZGRENZEIn : ITF_EINSATZGRENZE;	
END_VAR
    RoundedRectangle (1,1 820x700)
    RoundedRectangle (11,11 799x679)
    Frame (16,51 800x630), invisible if: NOT __QUERYINTERFACE(ITF_EINSATZGRENZEIn,ITF_EINSATZGRENZEIn)
        shows VIS_DIA_EINSATZGRENZE(fbEinsatzgrenzeIn := ITF_EINSATZGRENZEIn.proTHIS_REF)
    Image (761,10 50x50), image: CtaVisSymbols.ImagePool.close_solo_black
        OnMouseClick:  Dialog=DIA_EINSATZGRENZE, Result=OK, NumpadKeypadSet=True
    Label (21,16 730x30), "Parameter Einsatztdiagramm"
    InvisibleInput (11,1 750x48)
END_VISUALIZATION

// 40 Visualizations/EINSATZGRENZE/VIS_EINSATZGRENZE_ITF
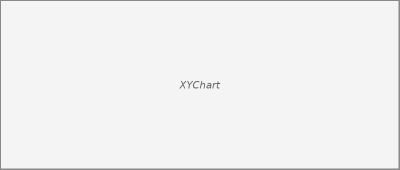
VISUALIZATION VIS_EINSATZGRENZE_ITF  // 400x170
VAR_INPUT
	fbEinsatzgrenzeIn : REFERENCE TO fbEinsatzgrenze;
END_VAR
    XYChart (0,0 400x170)
END_VISUALIZATION

// 40 Visualizations/EINSATZGRENZE/VIS_EINSATZGRENZE_QUERRY
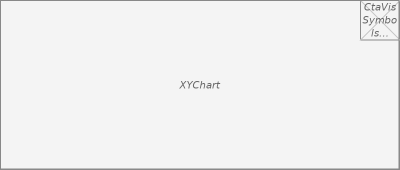
VISUALIZATION VIS_EINSATZGRENZE_QUERRY  // 400x170
VAR_INPUT
    {attribute 'initialize_on_call'}
    ITF_EINSATZGRENZEIn : ITF_EINSATZGRENZE;	
END_VAR
    Frame (0,0 400x170), invisible if: NOT __QUERYINTERFACE(ITF_EINSATZGRENZEIn,ITF_EINSATZGRENZEIn)
        shows VIS_EINSATZGRENZE_ITF(fbEinsatzgrenzeIn := ITF_EINSATZGRENZEIn.proTHIS_REF)
    Image (360,0 40x40), invisible if: NOT __QUERYINTERFACE(ITF_EINSATZGRENZEIn,ITF_EINSATZGRENZEIn), image: CtaVisSymbols.ImagePool.gear
        OnMouseClick:  Dialog=DIA_EINSATZGRENZE, Parameters={ITF_EINSATZGRENZEIn: ITF_EINSATZGRENZEIn}, OpenCentered=True
END_VISUALIZATION

// 40 Visualizations/EINSATZGRENZE/DIALOG/VIS_DIA_EINSATZGRENZE
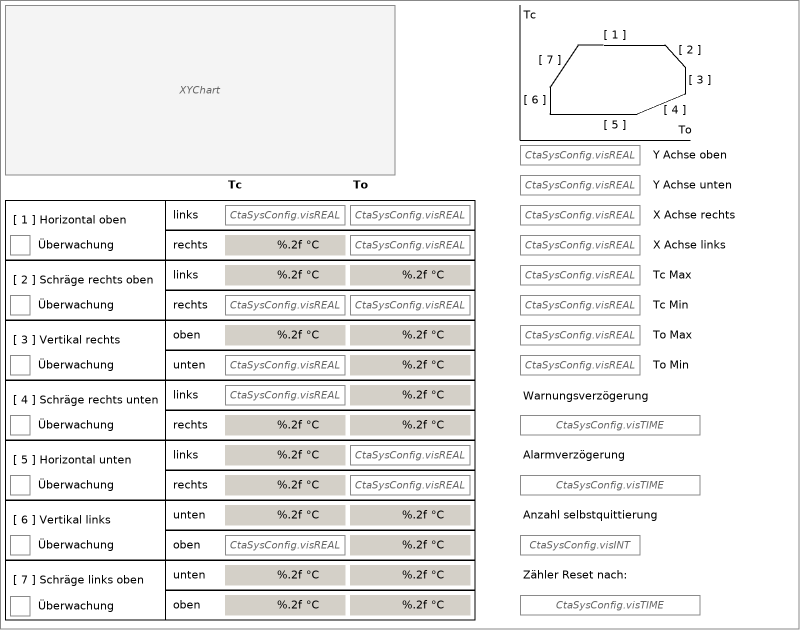
VISUALIZATION VIS_DIA_EINSATZGRENZE  // 800x630
VAR_INPUT
	fbEinsatzgrenzeIn : REFERENCE TO fbEinsatzgrenze;
END_VAR
    Frame (5,5 390x170)
        shows VIS_DIA_EINSATZGRENZE_ITF(fbEinsatzgrenzeIn := fbEinsatzgrenzeIn)
        p118247739: fbEinsatzgrenze
    Label (225,175 80x20), "Tc"
    Label (350,175 80x20), "To"
    Group (520,5 190x136)
        Group (5,20 185x110)
            Group (25,20 135x69)
                Polyline (54,0) (115,0) (135,22) (135,49) (87,69)
                Polyline (53,0) (28,0) (0,42) (0,69) (87,69)
            Label (80,0 20x20), "[ 1 ]"
            Label (155,15 20x20), "[ 2 ]"
            Label (165,45 20x20), "[ 3 ]"
            Label (140,75 20x20), "[ 4 ]"
            Label (80,90 20x20), "[ 5 ]"
            Label (0,65 20x20), "[ 6 ]"
            Label (15,25 20x20), "[ 7 ]"
        Label (0,0 20x20), "Tc"
        Label (155,115 20x20), "To"
        Line (0,135) (170,135)
        Line (0,135) (0,0)
    Group (520,145 210x470)
        Frame (0,120 120x20)
            shows CtaSysConfig.visREAL(visfbREALIn := fbEinsatzgrenzeIn.scParaData.fbrMaxTc, stPhysikalischeEinheit := '°C')
        Frame (0,150 120x20)
            shows CtaSysConfig.visREAL(visfbREALIn := fbEinsatzgrenzeIn.scParaData.fbrMinTc, stPhysikalischeEinheit := '°C')
        Frame (0,180 120x20)
            shows CtaSysConfig.visREAL(visfbREALIn := fbEinsatzgrenzeIn.scParaData.fbrMaxTo, stPhysikalischeEinheit := '°C')
        Frame (0,210 120x20)
            shows CtaSysConfig.visREAL(visfbREALIn := fbEinsatzgrenzeIn.scParaData.fbrMinTo, stPhysikalischeEinheit := '°C')
        Label (130,120 80x20), "Tc Max"
        Label (130,150 80x20), "Tc Min"
        Label (130,180 80x20), "To Max"
        Label (130,210 80x20), "To Min"
        Frame (0,330 180x20)
            shows CtaSysConfig.visTIME(visfbTIMEIn := fbEinsatzgrenzeIn.scParaData.scErrorWarning.fbtDelayError)
        Label (0,300 150x20), "Alarmverzögerung"
        Frame (0,270 180x20)
            shows CtaSysConfig.visTIME(visfbTIMEIn := fbEinsatzgrenzeIn.scParaData.scErrorWarning.fbtDelayWarning)
        Label (0,241 150x20), "Warnungsverzögerung"
        Frame (0,390 120x20)
            shows CtaSysConfig.visINT(visfbINTIn := fbEinsatzgrenzeIn.scParaData.scErrorWarning.fbiAnzError, stPhysikalischeEinheit := '')
        Frame (0,450 180x20)
            shows CtaSysConfig.visTIME(visfbTIMEIn := fbEinsatzgrenzeIn.scParaData.scErrorWarning.fbtCountReset)
        Label (0,420 150x20), "Zähler Reset nach:"
        Label (0,360 150x20), "Anzahl selbstquittierung"
        Frame (0,0 120x20)
            shows CtaSysConfig.visREAL(visfbREALIn := fbEinsatzgrenzeIn.scParaData.scDiagrammSize.fbrYMax, stPhysikalischeEinheit := '°C')
        Frame (0,30 120x20)
            shows CtaSysConfig.visREAL(visfbREALIn := fbEinsatzgrenzeIn.scParaData.scDiagrammSize.fbrYMin, stPhysikalischeEinheit := '°C')
        Frame (0,60 120x20)
            shows CtaSysConfig.visREAL(visfbREALIn := fbEinsatzgrenzeIn.scParaData.scDiagrammSize.fbrXMax, stPhysikalischeEinheit := '°C')
        Frame (0,90 120x20)
            shows CtaSysConfig.visREAL(visfbREALIn := fbEinsatzgrenzeIn.scParaData.scDiagrammSize.fbrXMin, stPhysikalischeEinheit := '°C')
        Label (130,0 80x20), "Y Achse oben"
        Label (130,30 80x20), "Y Achse unten"
        Label (130,60 80x20), "X Achse rechts"
        Label (130,90 80x20), "X Achse links"
    Group (5,200 470x420)
        Rectangle (0,0 470x60)
        Rectangle (160,0 310x30)
        Frame (220,5 120x20)
            shows CtaSysConfig.visREAL(visfbREALIn := fbEinsatzgrenzeIn.scParaData.scSlopValue1.fbrTcL, stPhysikalischeEinheit := '°C')
        Frame (345,5 120x20)
            shows CtaSysConfig.visREAL(visfbREALIn := fbEinsatzgrenzeIn.scParaData.scSlopValue1.fbrT0L, stPhysikalischeEinheit := '°C')
        Label (165,5 50x20), "links"
        Label (5,10 150x20), "[ 1 ] Horizontal oben"
        Rectangle (160,30 310x30)
        Frame (345,35 120x20)
            shows CtaSysConfig.visREAL(visfbREALIn := fbEinsatzgrenzeIn.scParaData.scSlopValue1.fbrT0R, stPhysikalischeEinheit := '°C')
        Textfield (220,35 80x20), "%.2f", text variable: fbEinsatzgrenzeIn.scParaData.scSlopValue1.fbrTcL.rValue
        Label (165,35 50x20), "rechts"
        Group (5,35 125x20)
            Frame (0,0 20x20)
                shows CtaSysConfig.visBOOL(visfbBOOLIn := fbEinsatzgrenzeIn.scParaData.scErrorWarning.fbxEnEW1)
            Label (25,0 100x20), "Überwachung"
        Rectangle (0,60 470x60)
        Label (5,70 150x20), "[ 2 ] Schräge rechts oben"
        Rectangle (160,90 310x30)
        Frame (220,95 120x20)
            shows CtaSysConfig.visREAL(visfbREALIn := fbEinsatzgrenzeIn.scParaData.scSlopValue2.fbrTcR, stPhysikalischeEinheit := '°C')
        Frame (345,95 120x20)
            shows CtaSysConfig.visREAL(visfbREALIn := fbEinsatzgrenzeIn.scParaData.scSlopValue2.fbrT0R, stPhysikalischeEinheit := '°C')
        Label (165,95 50x20), "rechts"
        Rectangle (160,60 310x30)
        Label (165,65 50x20), "links"
        Textfield (220,65 80x20), "%.2f", text variable: fbEinsatzgrenzeIn.scParaData.scSlopValue1.fbrTcL.rValue
        Textfield (345,65 80x20), "%.2f", text variable: fbEinsatzgrenzeIn.scParaData.scSlopValue1.fbrT0R.rValue
        Group (5,95 125x20)
            Frame (0,0 20x20)
                shows CtaSysConfig.visBOOL(visfbBOOLIn := fbEinsatzgrenzeIn.scParaData.scErrorWarning.fbxEnEW2)
            Label (25,0 100x20), "Überwachung"
        Rectangle (0,120 470x60)
        Label (5,130 150x20), "[ 3 ] Vertikal rechts"
        Rectangle (160,120 310x30)
        Label (165,125 50x20), "oben"
        Textfield (220,125 80x20), "%.2f", text variable: fbEinsatzgrenzeIn.scParaData.scSlopValue2.fbrTcR.rValue
        Textfield (345,125 80x20), "%.2f", text variable: fbEinsatzgrenzeIn.scParaData.scSlopValue2.fbrT0R.rValue
        Rectangle (160,150 310x30)
        Frame (220,155 120x20)
            shows CtaSysConfig.visREAL(visfbREALIn := fbEinsatzgrenzeIn.scParaData.scSlopValue3.fbrTcU, stPhysikalischeEinheit := '°C')
        Label (165,155 50x20), "unten"
        Textfield (345,155 80x20), "%.2f", text variable: fbEinsatzgrenzeIn.scParaData.scSlopValue2.fbrT0R.rValue
        Group (5,155 125x20)
            Frame (0,0 20x20)
                shows CtaSysConfig.visBOOL(visfbBOOLIn := fbEinsatzgrenzeIn.scParaData.scErrorWarning.fbxEnEW3)
            Label (25,0 100x20), "Überwachung"
        Rectangle (0,180 470x60)
        Label (5,190 150x20), "[ 4 ] Schräge rechts unten"
        Rectangle (160,180 310x30)
        Frame (220,185 120x20)
            shows CtaSysConfig.visREAL(visfbREALIn := fbEinsatzgrenzeIn.scParaData.scSlopValue4.fbrTcL, stPhysikalischeEinheit := '°C')
        Label (165,185 50x20), "links"
        Textfield (345,185 80x20), "%.2f", text variable: fbEinsatzgrenzeIn.scParaData.scSlopValue5.fbrT0L.rValue
        Rectangle (160,210 310x30)
        Textfield (220,215 80x20), "%.2f", text variable: fbEinsatzgrenzeIn.scParaData.scSlopValue3.fbrTcU.rValue
        Label (165,215 50x20), "rechts"
        Textfield (345,215 80x20), "%.2f", text variable: fbEinsatzgrenzeIn.scParaData.scSlopValue2.fbrT0R.rValue
        Group (5,215 125x20)
            Frame (0,0 20x20)
                shows CtaSysConfig.visBOOL(visfbBOOLIn := fbEinsatzgrenzeIn.scParaData.scErrorWarning.fbxEnEW4)
            Label (25,0 100x20), "Überwachung"
        Rectangle (0,240 470x60)
        Label (5,250 150x20), "[ 5 ] Horizontal unten"
        Rectangle (160,240 310x30)
        Frame (345,245 120x20), text variable: fbEinsatzgrenzeIn.scParaData.scSlopValue5.fbrT0L
            shows CtaSysConfig.visREAL(visfbREALIn := fbEinsatzgrenzeIn.scParaData.scSlopValue5.fbrT0L, stPhysikalischeEinheit := '°C')
        Label (165,245 50x20), "links"
        Textfield (220,245 80x20), "%.2f", text variable: fbEinsatzgrenzeIn.scParaData.scSlopValue4.fbrTcL.rValue
        Rectangle (160,270 310x30)
        Textfield (220,275 80x20), "%.2f", text variable: fbEinsatzgrenzeIn.scParaData.scSlopValue4.fbrTcL.rValue
        Label (165,275 50x20), "rechts"
        Frame (345,275 120x20)
            shows CtaSysConfig.visREAL(visfbREALIn := fbEinsatzgrenzeIn.scParaData.scSlopValue5.fbrT0R, stPhysikalischeEinheit := '°C')
        Group (5,275 125x20)
            Frame (0,0 20x20)
                shows CtaSysConfig.visBOOL(visfbBOOLIn := fbEinsatzgrenzeIn.scParaData.scErrorWarning.fbxEnEW5)
            Label (25,0 100x20), "Überwachung"
        Rectangle (0,300 470x60)
        Label (5,310 150x20), "[ 6 ] Vertikal links"
        Rectangle (160,330 310x30)
        Textfield (345,335 80x20), "%.2f", text variable: fbEinsatzgrenzeIn.scParaData.scSlopValue5.fbrT0L.rValue
        Label (165,335 50x20), "oben"
        Frame (220,335 120x20)
            shows CtaSysConfig.visREAL(visfbREALIn := fbEinsatzgrenzeIn.scParaData.scSlopValue6.fbrTcO, stPhysikalischeEinheit := '°C')
        Rectangle (160,300 310x30)
        Label (165,305 50x20), "unten"
        Textfield (220,305 80x20), "%.2f", text variable: fbEinsatzgrenzeIn.scParaData.scSlopValue4.fbrTcL.rValue
        Textfield (345,305 80x20), "%.2f", text variable: fbEinsatzgrenzeIn.scParaData.scSlopValue5.fbrT0L.rValue
        Group (5,335 125x20)
            Frame (0,0 20x20)
                shows CtaSysConfig.visBOOL(visfbBOOLIn := fbEinsatzgrenzeIn.scParaData.scErrorWarning.fbxEnEW6)
            Label (25,0 100x20), "Überwachung"
        Rectangle (0,360 470x60)
        Label (5,370 150x20), "[ 7 ] Schräge links oben"
        Rectangle (160,360 310x30)
        Label (165,365 50x20), "unten"
        Textfield (220,365 80x20), "%.2f", text variable: fbEinsatzgrenzeIn.scParaData.scSlopValue6.fbrTcO.rValue
        Textfield (345,365 80x20), "%.2f", text variable: fbEinsatzgrenzeIn.scParaData.scSlopValue5.fbrT0L.rValue
        Rectangle (160,390 310x30)
        Textfield (345,395 80x20), "%.2f", text variable: fbEinsatzgrenzeIn.scParaData.scSlopValue1.fbrT0L.rValue
        Label (165,395 50x20), "oben"
        Textfield (220,395 80x20), "%.2f", text variable: fbEinsatzgrenzeIn.scParaData.scSlopValue1.fbrTcL.rValue
        Group (5,396 125x20)
            Frame (0,0 20x20)
                shows CtaSysConfig.visBOOL(visfbBOOLIn := fbEinsatzgrenzeIn.scParaData.scErrorWarning.fbxEnEW7)
            Label (25,0 100x20), "Überwachung"
        Textfield (298,35 42x20), "°C", text variable: fbEinsatzgrenzeIn.scParaData.scSlopValue1.fbrTcL.rValue
        Textfield (298,65 42x20), "°C", text variable: fbEinsatzgrenzeIn.scParaData.scSlopValue1.fbrTcL.rValue
        Textfield (423,65 42x20), "°C", text variable: fbEinsatzgrenzeIn.scParaData.scSlopValue1.fbrTcL.rValue
        Textfield (298,125 42x20), "°C", text variable: fbEinsatzgrenzeIn.scParaData.scSlopValue1.fbrTcL.rValue
        Textfield (423,125 42x20), "°C", text variable: fbEinsatzgrenzeIn.scParaData.scSlopValue1.fbrTcL.rValue
        Textfield (423,155 42x20), "°C", text variable: fbEinsatzgrenzeIn.scParaData.scSlopValue1.fbrTcL.rValue
        Textfield (423,185 42x20), "°C", text variable: fbEinsatzgrenzeIn.scParaData.scSlopValue1.fbrTcL.rValue
        Textfield (423,215 42x20), "°C", text variable: fbEinsatzgrenzeIn.scParaData.scSlopValue1.fbrTcL.rValue
        Textfield (298,215 42x20), "°C", text variable: fbEinsatzgrenzeIn.scParaData.scSlopValue1.fbrTcL.rValue
        Textfield (298,245 42x20), "°C", text variable: fbEinsatzgrenzeIn.scParaData.scSlopValue1.fbrTcL.rValue
        Textfield (298,275 42x20), "°C", text variable: fbEinsatzgrenzeIn.scParaData.scSlopValue1.fbrTcL.rValue
        Textfield (298,305 42x20), "°C", text variable: fbEinsatzgrenzeIn.scParaData.scSlopValue1.fbrTcL.rValue
        Textfield (423,305 42x20), "°C", text variable: fbEinsatzgrenzeIn.scParaData.scSlopValue1.fbrTcL.rValue
        Textfield (423,335 42x20), "°C", text variable: fbEinsatzgrenzeIn.scParaData.scSlopValue1.fbrTcL.rValue
        Textfield (298,365 42x20), "°C", text variable: fbEinsatzgrenzeIn.scParaData.scSlopValue1.fbrTcL.rValue
        Textfield (423,365 42x20), "°C", text variable: fbEinsatzgrenzeIn.scParaData.scSlopValue1.fbrTcL.rValue
        Textfield (423,395 42x20), "°C", text variable: fbEinsatzgrenzeIn.scParaData.scSlopValue1.fbrTcL.rValue
        Textfield (298,395 42x20), "°C", text variable: fbEinsatzgrenzeIn.scParaData.scSlopValue1.fbrTcL.rValue
END_VISUALIZATION

// 40 Visualizations/EINSATZGRENZE/DIALOG/VIS_DIA_EINSATZGRENZE_ITF
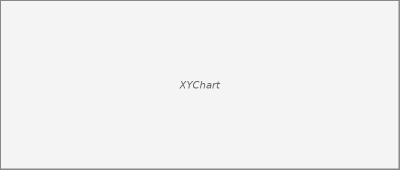
VISUALIZATION VIS_DIA_EINSATZGRENZE_ITF  // 400x170
VAR_INPUT
	fbEinsatzgrenzeIn : REFERENCE TO fbEinsatzgrenze;
END_VAR
VAR

END_VAR
    XYChart (0,0 400x170)
END_VISUALIZATION

(* text list Error (id | default | de | en | fr | it)
  11 | Einsatzgrenze, überschritten (oben) | Einsatzgrenze, überschritten (oben) | Application limit, exceeded (above) | Limite d'application, dépassée (en haut) | Limite di applicazione, superato (sopra)
  12 | Einsatzgrenze, überschritten (oben rechts) | Einsatzgrenze, überschritten (oben rechts) | Application limit, exceeded (top right) | Limite d'application, dépassée (en haut à droite) | Limite di applicazione, superato (sopra a destra)
  13 | Einsatzgrenze, überschritten (rechts) | Einsatzgrenze, überschritten (rechts) | Application limit, exceeded (right) | Limite d'application, dépassée (à droite) | Limite di applicazione, superato (a destra)
  14 | Einsatzgrenze, überschritten (unten rechts) | Einsatzgrenze, überschritten (unten rechts) | Application limit, exceeded (bottom right) | Limite d'application, dépassée (en bas à droite) | Limite di applicazione, superato (sotto a destra)
  15 | Einsatzgrenze, überschritten (unten) | Einsatzgrenze, überschritten (unten) | Application limit, exceeded (below) | Limite d'application, dépassée (en bas) | Limite di applicazione, superato (sotto)
  16 | Einsatzgrenze, überschritten (links) | Einsatzgrenze, überschritten (links) | Application limit, exceeded (left) | Limite d'application, dépassée (gauche) | Limite di applicazione, superato (sinistra)
  17 | Einsatzgrenze, überschritten (oben links) | Einsatzgrenze, überschritten (oben links) | Application limit, exceeded (top left) | Limite d'application, dépassée (en haut à gauche) | Limite di applicazione, superato (sopra a sinistra)
   |  |  |  |  |  *)

(* text list Info (id | default | de | en | fr | it)
  0 | keine Meldung Anstehend | keine Meldung Anstehend | no message pending | aucun message en attente | nessun messaggio in sospeso
   |  |  |  |  |  *)

(* text list Warnung (id | default | de | en | fr | it)
  11 | Einsatzgrenze, überschritten (oben) | Einsatzgrenze, überschritten (oben) | Application limit, exceeded (above) | Limite d'application, dépassée (en haut) | Limite di applicazione, superato (sopra)
  12 | Einsatzgrenze, überschritten (oben rechts) | Einsatzgrenze, überschritten (oben rechts) | Application limit, exceeded (top right) | Limite d'application, dépassée (en haut à droite) | Limite di applicazione, superato (sopra a destra)
  13 | Einsatzgrenze, überschritten (rechts) | Einsatzgrenze, überschritten (rechts) | Application limit, exceeded (right) | Limite d'application, dépassée (à droite) | Limite di applicazione, superato (a destra)
  14 | Einsatzgrenze, überschritten (unten rechts) | Einsatzgrenze, überschritten (unten rechts) | Application limit, exceeded (bottom right) | Limite d'application, dépassée (en bas à droite) | Limite di applicazione, superato (sotto a destra)
  15 | Einsatzgrenze, überschritten (unten) | Einsatzgrenze, überschritten (unten) | Application limit, exceeded (below) | Limite d'application, dépassée (en bas) | Limite di applicazione, superato (sotto)
  16 | Einsatzgrenze, überschritten (links) | Einsatzgrenze, überschritten (links) | Application limit, exceeded (left) | Limite d'application, dépassée (gauche) | Limite di applicazione, superato (sinistra)
  17 | Einsatzgrenze, überschritten (oben links) | Einsatzgrenze, überschritten (oben links) | Application limit, exceeded (top left) | Limite d'application, dépassée (en haut à gauche) | Limite di applicazione, superato (sopra a sinistra)
   |  |  |  |  |  *)
